{attribute 'GeneratedUsingTerminal: AT2050-0501-0023'}
{attribute addProperty BoxType "AT2050-0501-0023"}
{attribute addProperty Id "A_0083_AT2050_5500_0016_AT2050_5500AT2050_33A3DF1B80"}
{attribute addProperty CRC "2781648516"}
{attribute addProperty Size "80"}
TYPE A_0071_AT2050_0501_0023_AT2050_0501_A5CC9684 EXTENDS AT2050_2EA6C9BF :
STRUCT
	{attribute addProperty Name "A_0083_AT2050_5500_0016_AT2050_5500"}
	{attribute addProperty PreviousPort "A_0071(AT2050-0501-0023) (AT2050-0501) : B"}
	A_0083_AT2050_5500_0016_AT2050_5500 : AT2050_33A3DF1B;
END_STRUCT
END_TYPE

(* stored: Version 1.2.0.0, ProductVersion 3.1.4024.9
   DUT A_0071_AT2050_0501_0023_AT2050_0501_A5CC9684: Id {2ad561da-df88-4460-b4b6-a9d2726d1434} *)
